TYPE TcoQlSeriesSupply_Config_v_1_x_x : 
STRUCT
    InfoTime : TIME := T#2S;
    ErrorTime : TIME := T#0S;
    IpAddress : STRING;
    Port : UINT := 9221;
    Timeout : UINT := 1000;
END_STRUCT
END_TYPE

(* stored: Version 1.1.0.1, ProductVersion 3.1.4024.12
   DUT TcoQlSeriesSupply_Config_v_1_x_x: Id {56710dec-3679-0057-0877-f1de0cbea9ba} *)
